// C = A - B;
FUNCTION vecSub : BOOL
VAR_IN_OUT CONSTANT
	vecA :ARRAY[*] OF LREAL;
	vecB :ARRAY[*] OF LREAL;
END_VAR

VAR_IN_OUT 
	vecC :ARRAY[*] OF LREAL;
END_VAR

VAR
	m :DINT;
	i:DINT;
 
END_VAR

m:=UPPER_BOUND(VecA,1);

FOR i:=1 TO m DO
	vecC[i]:=vecA[i]-vecB[i];
END_FOR

END_FUNCTION

(* stored: Version 1.1.0.1, ProductVersion 3.1.4024.12
   POU vecSub: Id {1f77be5e-18b6-4c1a-b130-e7770100154c}, SpecialFunc None *)
